        // ===========================================
        // STEP 39: Axis_XToGlueSafPos_2
        // ===========================================
        STEP_ST10_Flow7_CGlueing_Axis_XToGlueSafPos_2:
            // Action Qualifier=N
            // Token: "IAI_DeviceCtl".IAIServo[#X_Axis].Point[2].Start
            "IAI_DeviceCtl".IAIServo[#X_Axis].Point[2].Start;

            // Transition to next step: 51
            IF TRUE THEN  // Sequential transition - review XML for actual condition
                #State := STEP_ST10_Flow7_CGlueing_TimeDelay_3;
            END_IF;

        // ===========================================
        // STEP 51: TimeDelay_3
        // ===========================================
        STEP_ST10_Flow7_CGlueing_TimeDelay_3:
            // No actions in XML

            // Transition to next step: 144
            IF TRUE THEN  // Sequential transition - review XML for actual condition
                #State := STEP_ST10_Flow7_CGlueing_ServoHomePos_6;
            END_IF;

        // ===========================================
        // STEP 144: ServoHomePos_6
        // ===========================================
        STEP_ST10_Flow7_CGlueing_ServoHomePos_6:
            // Action Qualifier=S
            // Token: "ServoV90_A3".IO.ioAutoHome
            "ServoV90_A3".IO.ioAutoHome := TRUE;

            // Transition to next step: 282
            IF TRUE THEN  // Sequential transition - review XML for actual condition
                #State := STEP_ST10_Flow7_CGlueing_RequestRobotGluePick;
            END_IF;

        // ===========================================
        // STEP 282: RequestRobotGluePick
        // ===========================================
        STEP_ST10_Flow7_CGlueing_RequestRobotGluePick:
            // Action Qualifier=N
            // Token: "AutoProcessControl".C_Glue.Robot2PickPrimit
            "AutoProcessControl".C_Glue.Robot2PickPrimit;

            // Transition to next step: 310
            IF TRUE THEN  // Sequential transition - review XML for actual condition
                #State := STEP_ST10_Flow7_CGlueing_MESCheckRequest;
            END_IF;

        // ===========================================
        // STEP 310: MESCheckRequest
        // ===========================================
        STEP_ST10_Flow7_CGlueing_MESCheckRequest:
            // Action Qualifier=N
            // Token: "PLCtoMES"."PLC.Load_Station5ChickInReq"
            "PLCtoMES"."PLC.Load_Station5ChickInReq";

            // Transition to next step: 78
            IF TRUE THEN  // Sequential transition - review XML for actual condition
                #State := STEP_ST10_Flow7_CGlueing_Axis_ZToIVCheckPos;
            END_IF;

        // ===========================================
        // STEP 78: Axis_ZToIVCheckPos
        // ===========================================
        STEP_ST10_Flow7_CGlueing_Axis_ZToIVCheckPos:
            // Action Qualifier=N
            // Token: "IAI_DeviceCtl".IAIServo[#Z_Axis].Point[7].Start
            "IAI_DeviceCtl".IAIServo[#Z_Axis].Point[7].Start;

            // Transition to next step: 329
            IF TRUE THEN  // Sequential transition - review XML for actual condition
                #State := STEP_ST10_Flow7_CGlueing_ok_1;
            END_IF;

        // ===========================================
        // STEP 329: ok_1
        // ===========================================
        STEP_ST10_Flow7_CGlueing_ok_1:
            // Action Qualifier=N
            // Token: "AutoProcessData".C_Glue.PartStatus := 399
            "AutoProcessData".C_Glue.PartStatus := 399;

            // Transition to next step: 30
            IF TRUE THEN  // Sequential transition - review XML for actual condition
                #State := STEP_ST10_Flow7_CGlueing_CheckGlueSysOK;
            END_IF;

        // ===========================================
        // STEP 30: CheckGlueSysOK
        // ===========================================
        STEP_ST10_Flow7_CGlueing_CheckGlueSysOK:
            // No actions in XML

            // Transition to next step: 108
            IF TRUE THEN  // Sequential transition - review XML for actual condition
                #State := STEP_ST10_Flow7_CGlueing_IAIMoveFinish_2;
            END_IF;

        // ===========================================
        // STEP 108: IAIMoveFinish_2
        // ===========================================
        STEP_ST10_Flow7_CGlueing_IAIMoveFinish_2:
            // No actions in XML

            // Transition to next step: 89
            IF TRUE THEN  // Sequential transition - review XML for actual condition
                #State := STEP_ST10_Flow7_CGlueing_Axis_ZToGlueePos_1;
            END_IF;

        // ===========================================
        // STEP 89: Axis_ZToGlueePos_1
        // ===========================================
        STEP_ST10_Flow7_CGlueing_Axis_ZToGlueePos_1:
            // Action Qualifier=N
            // Token: "IAI_DeviceCtl".IAIServo[#Z_Axis].Point[2].Start
            "IAI_DeviceCtl".IAIServo[#Z_Axis].Point[2].Start;

            // Transition to next step: 163
            IF TRUE THEN  // Sequential transition - review XML for actual condition
                #State := STEP_ST10_Flow7_CGlueing_Glue2s;
            END_IF;

        // ===========================================
        // STEP 163: Glue2s
        // ===========================================
        STEP_ST10_Flow7_CGlueing_Glue2s:
            // Action Qualifier=N
            // Token: "GluingControl".GlueInitiaStart
            "GluingControl".GlueInitiaStart;

            // Transition to next step: 94
            IF TRUE THEN  // Sequential transition - review XML for actual condition
                #State := STEP_ST10_Flow7_CGlueing_ServoHomePos;
            END_IF;

        // ===========================================
        // STEP 94: ServoHomePos
        // ===========================================
        STEP_ST10_Flow7_CGlueing_ServoHomePos:
            // Action Qualifier=S
            // Token: "ServoV90_A3".IO.ioAutoHome
            "ServoV90_A3".IO.ioAutoHome := TRUE;

            // Transition to next step: 35
            IF TRUE THEN  // Sequential transition - review XML for actual condition
                #State := STEP_ST10_Flow7_CGlueing_Axis_ZToGlueePos_2;
            END_IF;

        // ===========================================
        // STEP 35: Axis_ZToGlueePos_2
        // ===========================================
        STEP_ST10_Flow7_CGlueing_Axis_ZToGlueePos_2:
            // Action Qualifier=N
            // Token: "IAI_DeviceCtl".IAIServo[#Z_Axis].Point[3].Start
            "IAI_DeviceCtl".IAIServo[#Z_Axis].Point[3].Start;

            // Transition to next step: 60
            IF TRUE THEN  // Sequential transition - review XML for actual condition
                #State := STEP_ST10_Flow7_CGlueing_IV3Check;
            END_IF;

        // ===========================================
        // STEP 60: IV3Check
        // ===========================================
        STEP_ST10_Flow7_CGlueing_IV3Check:
            // Action Qualifier=N, Event="S1"
            // Token: "DB_KeyenceCheckerIV3".aDev[2].Common.nMode := 1
            "DB_KeyenceCheckerIV3".aDev[2].Common.nMode := 1;

            // Transition to next step: 110
            IF TRUE THEN  // Sequential transition - review XML for actual condition
                #State := STEP_ST10_Flow7_CGlueing_Step110;
            END_IF;

        // ===========================================
        // STEP 110: Step110
        // ===========================================
        STEP_ST10_Flow7_CGlueing_Step110:
            // No actions in XML

            // Transition to next step: 65
            IF TRUE THEN  // Sequential transition - review XML for actual condition
                #State := STEP_ST10_Flow7_CGlueing_Magnet_Glue;
            END_IF;

        // ===========================================
        // STEP 65: Magnet_Glue
        // ===========================================
        STEP_ST10_Flow7_CGlueing_Magnet_Glue:
            // No actions in XML

            // Transition to next step: 48
            IF TRUE THEN  // Sequential transition - review XML for actual condition
                #State := STEP_ST10_Flow7_CGlueing_Servo_returns_toGluePos_3;
            END_IF;

        // ===========================================
        // STEP 48: Servo returns toGluePos_3
        // ===========================================
        STEP_ST10_Flow7_CGlueing_Servo_returns_toGluePos_3:
            // Action Qualifier=N
            // Token: "ServoV90_DeviceCtl".V90Servo[3].Point[4].Start
            "ServoV90_DeviceCtl".V90Servo[3].Point[4].Start;

            // Transition to next step: 112
            IF TRUE THEN  // Sequential transition - review XML for actual condition
                #State := STEP_ST10_Flow7_CGlueing_WaitIAIStop_3;
            END_IF;

        // ===========================================
        // STEP 112: WaitIAIStop_3
        // ===========================================
        STEP_ST10_Flow7_CGlueing_WaitIAIStop_3:
            // No actions in XML

            // Transition to next step: 326
            IF TRUE THEN  // Sequential transition - review XML for actual condition
                #State := STEP_ST10_Flow7_CGlueing_ResultNG;
            END_IF;

        // ===========================================
        // STEP 326: ResultNG
        // ===========================================
        STEP_ST10_Flow7_CGlueing_ResultNG:
            // Action Qualifier=N
            // Token: "AutoProcessData".C_Glue.PartStatus := 352
            "AutoProcessData".C_Glue.PartStatus := 352;

            // Transition to next step: 130
            IF TRUE THEN  // Sequential transition - review XML for actual condition
                #State := STEP_ST10_Flow7_CGlueing_NGStatus_2;
            END_IF;

        // ===========================================
        // STEP 130: NGStatus_2
        // ===========================================
        STEP_ST10_Flow7_CGlueing_NGStatus_2:
            // Action Qualifier=N
            // Token: "AutoProcessData".C_Glue.PartStatus := 359
            "AutoProcessData".C_Glue.PartStatus := 359;
            // Action Qualifier=N
            // Token: "Station5UnLoadData"."PLC.ShaftGlueIVScore2" := "DB_KeyenceCheckerIV3".aDev[2].In.ToolResult[2].nToolMatchingRate
            "Station5UnLoadData"."PLC.ShaftGlueIVScore2" := "DB_KeyenceCheckerIV3".aDev[2].In.ToolResult[2].nToolMatchingRate;
            // Action Qualifier=N
            // Token: "AutoProcessData".C_Glue.IV3_ShaftScore_2 := "DB_KeyenceCheckerIV3".aDev[2].In.ToolResult[2].nToolMatchingRate
            "AutoProcessData".C_Glue.IV3_ShaftScore_2 := "DB_KeyenceCheckerIV3".aDev[2].In.ToolResult[2].nToolMatchingRate;
            // Action Qualifier=N
            // Token: "AutoProcessData".C_Glue.IV3_ShaftCheckResult := 2
            "AutoProcessData".C_Glue.IV3_ShaftCheckResult := 2;

            // Transition to next step: 42
            IF TRUE THEN  // Sequential transition - review XML for actual condition
                #State := STEP_ST10_Flow7_CGlueing_TimeDelay_1;
            END_IF;

        // ===========================================
        // STEP 42: TimeDelay_1
        // ===========================================
        STEP_ST10_Flow7_CGlueing_TimeDelay_1:
            // No actions in XML

            // Transition to next step: 315
            IF TRUE THEN  // Sequential transition - review XML for actual condition
                #State := STEP_ST10_Flow7_CGlueing_Bypass;
            END_IF;

        // ===========================================
        // STEP 315: Bypass
        // ===========================================
        STEP_ST10_Flow7_CGlueing_Bypass:
            // No actions in XML

            // Transition to next step: 155
            IF TRUE THEN  // Sequential transition - review XML for actual condition
                #State := STEP_ST10_Flow7_CGlueing_IAIMoveFinish_4;
            END_IF;

        // ===========================================
        // STEP 155: IAIMoveFinish_4
        // ===========================================
        STEP_ST10_Flow7_CGlueing_IAIMoveFinish_4:
            // No actions in XML

            // Transition to next step: 208
            IF TRUE THEN  // Sequential transition - review XML for actual condition
                #State := STEP_ST10_Flow7_CGlueing_CheckIV3Ready_4;
            END_IF;

        // ===========================================
        // STEP 208: CheckIV3Ready_4
        // ===========================================
        STEP_ST10_Flow7_CGlueing_CheckIV3Ready_4:
            // Action Qualifier=N
            // Token: "DB_KeyenceCheckerIV3".aDev[2].Para.nProgramNo := 1
            "DB_KeyenceCheckerIV3".aDev[2].Para.nProgramNo := 1;

            // Transition to next step: 299
            IF TRUE THEN  // Sequential transition - review XML for actual condition
                #State := STEP_ST10_Flow7_CGlueing_ShaftGlueProcessFinish;
            END_IF;

        // ===========================================
        // STEP 299: ShaftGlueProcessFinish
        // ===========================================
        STEP_ST10_Flow7_CGlueing_ShaftGlueProcessFinish:
            // No actions in XML

            // Transition to next step: 106
            IF TRUE THEN  // Sequential transition - review XML for actual condition
                #State := STEP_ST10_Flow7_CGlueing_WaitIAIStop_1;
            END_IF;

        // ===========================================
        // STEP 106: WaitIAIStop_1
        // ===========================================
        STEP_ST10_Flow7_CGlueing_WaitIAIStop_1:
            // No actions in XML

            // Transition to next step: 317
            IF TRUE THEN  // Sequential transition - review XML for actual condition
                #State := STEP_ST10_Flow7_CGlueing_Check_NG;
            END_IF;

        // ===========================================
        // STEP 317: Check NG
        // ===========================================
        STEP_ST10_Flow7_CGlueing_Check_NG:
            // Action Qualifier=N
            // Token: "AutoProcessData".C_Glue.PartStatus := 351
            "AutoProcessData".C_Glue.PartStatus := 351;

            // Transition to next step: 76
            IF TRUE THEN  // Sequential transition - review XML for actual condition
                #State := STEP_ST10_Flow7_CGlueing_TimeDelay_5;
            END_IF;

        // ===========================================
        // STEP 76: TimeDelay_5
        // ===========================================
        STEP_ST10_Flow7_CGlueing_TimeDelay_5:
            // No actions in XML

            // Transition to next step: 22
            IF TRUE THEN  // Sequential transition - review XML for actual condition
                #State := STEP_ST10_Flow7_CGlueing_Servo_returns_toHome_Pos;
            END_IF;

        // ===========================================
        // STEP 22: Servo returns toHome Pos
        // ===========================================
        STEP_ST10_Flow7_CGlueing_Servo_returns_toHome_Pos:
            // Action Qualifier=N
            // Token: "ServoV90_DeviceCtl".V90Servo[3].Point[1].Start
            "ServoV90_DeviceCtl".V90Servo[3].Point[1].Start;

            // Transition to next step: 115
            IF TRUE THEN  // Sequential transition - review XML for actual condition
                #State := STEP_ST10_Flow7_CGlueing_ServoHomePos_3;
            END_IF;

        // ===========================================
        // STEP 115: ServoHomePos_3
        // ===========================================
        STEP_ST10_Flow7_CGlueing_ServoHomePos_3:
            // Action Qualifier=S
            // Token: "ServoV90_A3".IO.ioAutoHome
            "ServoV90_A3".IO.ioAutoHome := TRUE;

            // Transition to next step: 126
            IF TRUE THEN  // Sequential transition - review XML for actual condition
                #State := STEP_ST10_Flow7_CGlueing_CameraCheck2;
            END_IF;

        // ===========================================
        // STEP 126: CameraCheck2
        // ===========================================
        STEP_ST10_Flow7_CGlueing_CameraCheck2:
            // No actions in XML

            // Transition to next step: 28
            IF TRUE THEN  // Sequential transition - review XML for actual condition
                #State := STEP_ST10_Flow7_CGlueing_WaitRobot1FinishTask;
            END_IF;

        // ===========================================
        // STEP 28: WaitRobot1FinishTask
        // ===========================================
        STEP_ST10_Flow7_CGlueing_WaitRobot1FinishTask:
            // No actions in XML

            // Transition to next step: 162
            IF TRUE THEN  // Sequential transition - review XML for actual condition
                #State := STEP_ST10_Flow7_CGlueing_bypassGlue4;
            END_IF;

        // ===========================================
        // STEP 162: bypassGlue4
        // ===========================================
        STEP_ST10_Flow7_CGlueing_bypassGlue4:
            // No actions in XML

            // Transition to next step: 139
            IF TRUE THEN  // Sequential transition - review XML for actual condition
                #State := STEP_ST10_Flow7_CGlueing_IV3Check_4;
            END_IF;

        // ===========================================
        // STEP 139: IV3Check_4
        // ===========================================
        STEP_ST10_Flow7_CGlueing_IV3Check_4:
            // Action Qualifier=N, Event="S1"
            // Token: "DB_KeyenceCheckerIV3".aDev[2].Common.nMode := 1
            "DB_KeyenceCheckerIV3".aDev[2].Common.nMode := 1;

            // Transition to next step: 630
            IF TRUE THEN  // Sequential transition - review XML for actual condition
                #State := STEP_ST10_Flow7_CGlueing_IV3_Check;
            END_IF;

        // ===========================================
        // STEP 630: IV3 Check
        // ===========================================
        STEP_ST10_Flow7_CGlueing_IV3_Check:
            // No actions in XML

            // Transition to next step: 307
            IF TRUE THEN  // Sequential transition - review XML for actual condition
                #State := STEP_ST10_Flow7_CGlueing_Prepare_MES_CheckData_1;
            END_IF;

        // ===========================================
        // STEP 307: Prepare MES CheckData_1
        // ===========================================
        STEP_ST10_Flow7_CGlueing_Prepare_MES_CheckData_1:
            // No actions in XML

            // Transition to next step: 320
            IF TRUE THEN  // Sequential transition - review XML for actual condition
                #State := STEP_ST10_Flow7_CGlueing_MaganetGlue;
            END_IF;

        // ===========================================
        // STEP 320: MaganetGlue
        // ===========================================
        STEP_ST10_Flow7_CGlueing_MaganetGlue:
            // No actions in XML

            // Transition to next step: 109
            IF TRUE THEN  // Sequential transition - review XML for actual condition
                #State := STEP_ST10_Flow7_CGlueing_WaitIAIStop_2;
            END_IF;

        // ===========================================
        // STEP 109: WaitIAIStop_2
        // ===========================================
        STEP_ST10_Flow7_CGlueing_WaitIAIStop_2:
            // No actions in XML

            // Transition to next step: 32
            IF TRUE THEN  // Sequential transition - review XML for actual condition
                #State := STEP_ST10_Flow7_CGlueing_Axis_XToGlueSafPos;
            END_IF;

        // ===========================================
        // STEP 32: Axis_XToGlueSafPos
        // ===========================================
        STEP_ST10_Flow7_CGlueing_Axis_XToGlueSafPos:
            // Action Qualifier=N
            // Token: "IAI_DeviceCtl".IAIServo[#X_Axis].Point[2].Start
            "IAI_DeviceCtl".IAIServo[#X_Axis].Point[2].Start;

            // Transition to next step: 154
            IF TRUE THEN  // Sequential transition - review XML for actual condition
                #State := STEP_ST10_Flow7_CGlueing_IAIMoveFinish_5;
            END_IF;

        // ===========================================
        // STEP 154: IAIMoveFinish_5
        // ===========================================
        STEP_ST10_Flow7_CGlueing_IAIMoveFinish_5:
            // No actions in XML

            // Transition to next step: 203
            IF TRUE THEN  // Sequential transition - review XML for actual condition
                #State := STEP_ST10_Flow7_CGlueing_Total_Score_of_Shaft_Gluening_check;
            END_IF;

        // ===========================================
        // STEP 203: Total Score of Shaft Gluening check
        // ===========================================
        STEP_ST10_Flow7_CGlueing_Total_Score_of_Shaft_Gluening_check:
            // No actions in XML

            // Transition to next step: 21
            IF TRUE THEN  // Sequential transition - review XML for actual condition
                #State := STEP_ST10_Flow7_CGlueing_Axis_YToHomePos;
            END_IF;

        // ===========================================
        // STEP 21: Axis_YToHomePos
        // ===========================================
        STEP_ST10_Flow7_CGlueing_Axis_YToHomePos:
            // Action Qualifier=N
            // Token: "IAI_DeviceCtl".IAIServo[#Y_axis].Point[1].Start
            "IAI_DeviceCtl".IAIServo[#Y_axis].Point[1].Start;

            // Transition to next step: 43
            IF TRUE THEN  // Sequential transition - review XML for actual condition
                #State := STEP_ST10_Flow7_CGlueing_TimeDelay_2;
            END_IF;

        // ===========================================
        // STEP 43: TimeDelay_2
        // ===========================================
        STEP_ST10_Flow7_CGlueing_TimeDelay_2:
            // No actions in XML

            // Transition to next step: 145
            IF TRUE THEN  // Sequential transition - review XML for actual condition
                #State := STEP_ST10_Flow7_CGlueing_Step145;
            END_IF;

        // ===========================================
        // STEP 145: Step145
        // ===========================================
        STEP_ST10_Flow7_CGlueing_Step145:
            // No actions in XML

            // Transition to next step: 147
            IF TRUE THEN  // Sequential transition - review XML for actual condition
                #State := STEP_ST10_Flow7_CGlueing_CheckAxisXPos;
            END_IF;

        // ===========================================
        // STEP 147: CheckAxisXPos
        // ===========================================
        STEP_ST10_Flow7_CGlueing_CheckAxisXPos:
            // No actions in XML

            // Transition to next step: 119
            IF TRUE THEN  // Sequential transition - review XML for actual condition
                #State := STEP_ST10_Flow7_CGlueing_C_LocationCylinderToHP;
            END_IF;

        // ===========================================
        // STEP 119: C-LocationCylinderToHP
        // ===========================================
        STEP_ST10_Flow7_CGlueing_C_LocationCylinderToHP:
            // Action Qualifier=S
            // Token: "ST10Cylinder".Cy[9].Inout.AutoGoHome
            "ST10Cylinder".Cy[9].Inout.AutoGoHome := TRUE;
            // Action Qualifier=R
            // Token: "ST10Cylinder".Cy[9].Inout.AutoGoWork
            "ST10Cylinder".Cy[9].Inout.AutoGoWork := FALSE;

            // Transition to next step: 84
            IF TRUE THEN  // Sequential transition - review XML for actual condition
                #State := STEP_ST10_Flow7_CGlueing_OKStatus_1;
            END_IF;

        // ===========================================
        // STEP 84: OKStatus_1
        // ===========================================
        STEP_ST10_Flow7_CGlueing_OKStatus_1:
            // Action Qualifier=N
            // Token: "AutoProcessData".C_Glue.PartStatus := 380
            "AutoProcessData".C_Glue.PartStatus := 380;
            // Action Qualifier=N
            // Token: "Station5UnLoadData"."PLC.MagnetIVScore" := "DB_KeyenceCheckerIV3".aDev[1].In.ToolResult[2].nToolMatchingRate
            "Station5UnLoadData"."PLC.MagnetIVScore" := "DB_KeyenceCheckerIV3".aDev[1].In.ToolResult[2].nToolMatchingRate;
            // Action Qualifier=N
            // Token: "AutoProcessData".C_Glue.IV3_MagnetScore := "DB_KeyenceCheckerIV3".aDev[1].In.ToolResult[2].nToolMatchingRate
            "AutoProcessData".C_Glue.IV3_MagnetScore := "DB_KeyenceCheckerIV3".aDev[1].In.ToolResult[2].nToolMatchingRate;
            // Action Qualifier=N
            // Token: "AutoProcessData".C_Glue.IV3_MagnetCheckResult := 1
            "AutoProcessData".C_Glue.IV3_MagnetCheckResult := 1;

            // Transition to next step: 205
            IF TRUE THEN  // Sequential transition - review XML for actual condition
                #State := STEP_ST10_Flow7_CGlueing_Step204;
            END_IF;

        // ===========================================
        // STEP 205: Step204
        // ===========================================
        STEP_ST10_Flow7_CGlueing_Step204:
            // No actions in XML

            // Transition to next step: 107
            IF TRUE THEN  // Sequential transition - review XML for actual condition
                #State := STEP_ST10_Flow7_CGlueing_Step107;
            END_IF;

        // ===========================================
        // STEP 107: Step107
        // ===========================================
        STEP_ST10_Flow7_CGlueing_Step107:
            // No actions in XML

            // Transition to next step: 290
            IF TRUE THEN  // Sequential transition - review XML for actual condition
                #State := STEP_ST10_Flow7_CGlueing_Process__Finish;
            END_IF;

        // ===========================================
        // STEP 290: Process  Finish
        // ===========================================
        STEP_ST10_Flow7_CGlueing_Process__Finish:
            // Action Qualifier=S
            // Token: #ioPM_Inface.ProcessComplete
            #ioPM_Inface.ProcessComplete := TRUE;
            // Action Qualifier=R
            // Token: #ioPM_Inface.ProcessStart
            #ioPM_Inface.ProcessStart := FALSE;

            // Transition to next step: 58
            IF TRUE THEN  // Sequential transition - review XML for actual condition
                #State := STEP_ST10_Flow7_CGlueing_Glue_4;
            END_IF;

        // ===========================================
        // STEP 58: Glue_4
        // ===========================================
        STEP_ST10_Flow7_CGlueing_Glue_4:
            // No actions in XML

            // Transition to next step: 33
            IF TRUE THEN  // Sequential transition - review XML for actual condition
                #State := STEP_ST10_Flow7_CGlueing_Glue_1;
            END_IF;

        // ===========================================
        // STEP 33: Glue_1
        // ===========================================
        STEP_ST10_Flow7_CGlueing_Glue_1:
            // No actions in XML

            // Transition to next step: 133
            IF TRUE THEN  // Sequential transition - review XML for actual condition
                #State := STEP_ST10_Flow7_CGlueing_IV3Check_3;
            END_IF;

        // ===========================================
        // STEP 133: IV3Check_3
        // ===========================================
        STEP_ST10_Flow7_CGlueing_IV3Check_3:
            // Action Qualifier=N, Event="S1"
            // Token: "DB_KeyenceCheckerIV3".aDev[2].Common.nMode := 1
            "DB_KeyenceCheckerIV3".aDev[2].Common.nMode := 1;

            // Transition to next step: 66
            IF TRUE THEN  // Sequential transition - review XML for actual condition
                #State := STEP_ST10_Flow7_CGlueing_Magnet_GlueCheck;
            END_IF;

        // ===========================================
        // STEP 66: Magnet_GlueCheck
        // ===========================================
        STEP_ST10_Flow7_CGlueing_Magnet_GlueCheck:
            // No actions in XML

            // Transition to next step: 8
            IF TRUE THEN  // Sequential transition - review XML for actual condition
                #State := STEP_ST10_Flow7_CGlueing_WaitRobotInitialFinish;
            END_IF;

        // ===========================================
        // STEP 8: WaitRobotInitialFinish
        // ===========================================
        STEP_ST10_Flow7_CGlueing_WaitRobotInitialFinish:
            // No actions in XML

            // Transition to next step: 2
            IF TRUE THEN  // Sequential transition - review XML for actual condition
                #State := STEP_ST10_Flow7_CGlueing_S2;
            END_IF;

        // ===========================================
        // STEP 2: S2
        // ===========================================
        STEP_ST10_Flow7_CGlueing_S2:
            // No actions in XML

            // Transition to next step: 29
            IF TRUE THEN  // Sequential transition - review XML for actual condition
                #State := STEP_ST10_Flow7_CGlueing_Axis_XToGluePos_1;
            END_IF;

        // ===========================================
        // STEP 29: Axis_XToGluePos_1
        // ===========================================
        STEP_ST10_Flow7_CGlueing_Axis_XToGluePos_1:
            // Action Qualifier=N
            // Token: "IAI_DeviceCtl".IAIServo[#X_Axis].Point[3].Start
            "IAI_DeviceCtl".IAIServo[#X_Axis].Point[3].Start;

    END_CASE;

    // UPDATE ioPM_Inface
    #ioPM_Inface.InitialRun := #act_InitialRun;
    #ioPM_Inface.InitialOK := #act_InitialOK;
    #ioPM_Inface.WaitRunning := #act_WaitRunning;
    #ioPM_Inface.Running := #act_Running;
    #ioPM_Inface.ProcessComplete := #act_ProcessComplete;
    #ioPM_Inface.ProcessStart := #act_ProcessStart;
    #ioPM_Inface.UnPause := #act_UnPause;

    // ERROR HANDLING
    IF #bError THEN
        #ioStatus := 900;
        #oAlarmID := INT_TO_WORD(#wErrorID);
    ELSE
        #ioStatus := 0;
        #oAlarmID := 0;
    END_IF;
END_FUNCTION_BLOCK

//=============================================================================
// END OF FILE
//=============================================================================
